PROGRAM MAIN
VAR
	nisse: INT;
END_VAR

nisse:=nisse+1;

END_PROGRAM

(* stored: Version 1.1.0.1, ProductVersion 3.1.4024.13
   POU MAIN: Id {fbc17a05-003d-431c-bcdc-3161c0370a21}, SpecialFunc None *)
